Staubli VAL3: OnF6.pgx

program OnF6()
  local string l_sProperty[4]
  local string l_sItem
begin
  //
  l_sProperty[0]="工具"
  l_sProperty[1]="坐标系"
  l_sProperty[2]="安全点"
  l_sProperty[3]="可用点"
  call user:SetProerty("",26,7,6,4,l_sProperty,l_sItem)
  if l_sItem=="工具"
    Tool:libLoad("Tool")
    call Tool:Main(0)
    Tool:$libClose()
  elseIf l_sItem=="坐标系"
    Frame:libLoad("Frame")
    call Frame:start()
    Frame:$libClose()
  elseIf l_sItem=="安全点"
    Home:libLoad("Home")
    call Home:start()
    Home:$libClose()
  else
    SparePoint:libLoad("SparePoint")
    call SparePoint:start()
    SparePoint:$libClose()
  endIf
  bUserRefresh=true
end
